RESOURCE_TYPE _WaterHeaterController
  (* Standard: 61499-2 *)
  (* Version 0.1, 2017-00-25, hpea485, UOA *)
END_RESOURCE_TYPE
